# EPICS substitutions: pimegaApp/Db/pimega45d.substitutions
file "pimega.template" {
  {}
}

file "module.template" {
   pattern { MODULE, ADDR }
           { M1:,    0    }
}
